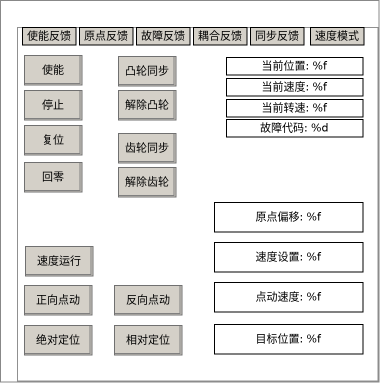
VISUALIZATION Vis_Axis  // 380x383
VAR_IN_OUT
	Axis:REFERENCE TO UDT_axisAdmin;
END_VAR
    GroupBox (17,19 361x362)
        Button (7,36 58x30), "使能"
            toggle Axis.i.Enable
        Button (8,227 68x30), "速度运行"
            tap Axis.i.MoveVel
        Button (101,37 58x30), "凸轮同步"
            tap Axis.i.CamIn
        Button (101,71 58x30), "解除凸轮"
            tap Axis.i.CamOut
        Button (7,71 58x30), "停止"
            tap Axis.i.Stop
        Button (7,106 58x30), "复位"
            tap Axis.i.Reset
        RoundedRectangle (209,38 137x18), "当前位置: %f", text variable: Axis.o.ActPos
        Button (7,266 68x30), "正向点动"
            tap Axis.i.JogP
        Button (97,266 68x30), "反向点动"
            tap Axis.i.JogN
        Rectangle (5,8 54x18), "使能反馈", colour toggle: Axis.o.PowerOn
        Rectangle (62,8 54x18), "原点反馈", colour toggle: Axis.o.Homed
        Rectangle (119,8 54x18), "故障反馈", colour toggle: Axis.o.Error
        Rectangle (176,8 54x18), "耦合反馈", colour toggle: Axis.o.InGear
        Rectangle (233,8 54x18), "同步反馈", colour toggle: Axis.o.InSync'
        Rectangle (293,8 54x18), "速度模式", colour toggle: Axis.o.InVelocity
        RoundedRectangle (209,59 137x18), "当前速度: %f", text variable: Axis.o.ActVel
        RoundedRectangle (209,80 137x18), "当前转速: %f", text variable: Axis.o.ActTorq
        Button (7,306 68x30), "绝对定位"
            tap Axis.i.MoveAbs
        Button (97,306 68x30), "相对定位"
            tap Axis.i.MoveAdd
        RoundedRectangle (197,263 149x30), "点动速度: %f", text variable: Axis.i.JogVel
            OnMouseClick: write the text variable via Default
        RoundedRectangle (197,305 149x30), "目标位置: %f", text variable: Axis.i.Pos
            OnMouseClick: write the text variable via Default
        RoundedRectangle (197,223 149x30), "速度设置: %f", text variable: Axis.i.Vel
            OnMouseClick: write the text variable via Default
        Button (101,148 58x30), "解除齿轮"
            tap Axis.i.GearOut
        RoundedRectangle (209,100 137x18), "故障代码: %d", text variable: Axis.o.ErrorID
        Button (7,143 58x30), "回零"
            tap Axis.i.Home
        RoundedRectangle (197,183 149x30), "原点偏移: %f", text variable: Axis.i.HomeOffset
            OnMouseClick: write the text variable via Default
    Button (118,133 58x30), "齿轮同步"
        tap Axis.i.GearIn
END_VISUALIZATION

(* stored: Version 1.1.0.1, ProductVersion 3.1.4022.16
   Visu Vis_Axis: Id {72456d0e-101d-46b0-a7b9-a4f5cf9a109d} *)
